  PROC DrawPart102()
    MoveL Offs(pOrigin,206.44,37.94,0.00),v40,z0,tPen\WObj:=wPaper;
    MoveL Offs(pOrigin,207.07,38.36,0.00),v40,z0,tPen\WObj:=wPaper;
    MoveL Offs(pOrigin,206.44,37.94,0.00),v40,fine,tPen\WObj:=wPaper;
    MoveL Offs(pOrigin,206.44,37.94,6.00),v60,z5,tPen\WObj:=wPaper;
    MoveL Offs(pOrigin,207.71,38.79,6.00),vTravel,z5,tPen\WObj:=wPaper;
    MoveL Offs(pOrigin,207.71,38.79,0.00),v60,z0,tPen\WObj:=wPaper;
    MoveL Offs(pOrigin,208.14,39.21,0.00),v40,z0,tPen\WObj:=wPaper;
    MoveL Offs(pOrigin,207.71,38.79,0.00),v40,z0,tPen\WObj:=wPaper;
    MoveL Offs(pOrigin,208.35,39.42,0.00),v40,z0,tPen\WObj:=wPaper;
    MoveL Offs(pOrigin,209.20,40.06,0.00),v40,z0,tPen\WObj:=wPaper;
    MoveL Offs(pOrigin,208.35,39.42,0.00),v40,fine,tPen\WObj:=wPaper;
    MoveL Offs(pOrigin,208.35,39.42,6.00),v60,z5,tPen\WObj:=wPaper;
    MoveL Offs(pOrigin,207.50,40.28,6.00),vTravel,z5,tPen\WObj:=wPaper;
    MoveL Offs(pOrigin,207.50,40.28,0.00),v60,z0,tPen\WObj:=wPaper;
    MoveL Offs(pOrigin,208.14,40.91,0.00),v40,z0,tPen\WObj:=wPaper;
    MoveL Offs(pOrigin,207.50,40.28,0.00),v40,fine,tPen\WObj:=wPaper;
    MoveL Offs(pOrigin,207.50,40.28,6.00),v60,z5,tPen\WObj:=wPaper;
    MoveL Offs(pOrigin,209.41,40.28,6.00),vTravel,z5,tPen\WObj:=wPaper;
    MoveL Offs(pOrigin,209.41,40.28,0.00),v60,z0,tPen\WObj:=wPaper;
    MoveL Offs(pOrigin,209.62,40.70,0.00),v40,z0,tPen\WObj:=wPaper;
    MoveL Offs(pOrigin,209.41,40.28,0.00),v40,fine,tPen\WObj:=wPaper;
    MoveL Offs(pOrigin,209.41,40.28,6.00),v60,z5,tPen\WObj:=wPaper;
    MoveL Offs(pOrigin,209.20,20.51,6.00),vTravel,z5,tPen\WObj:=wPaper;
    MoveL Offs(pOrigin,209.20,20.51,0.00),v60,z0,tPen\WObj:=wPaper;
    MoveL Offs(pOrigin,208.21,19.24,0.00),v40,z0,tPen\WObj:=wPaper;
    MoveL Offs(pOrigin,207.71,17.54,0.00),v40,z0,tPen\WObj:=wPaper;
    MoveL Offs(pOrigin,207.71,16.48,0.00),v40,z0,tPen\WObj:=wPaper;
    MoveL Offs(pOrigin,208.35,14.77,0.00),v40,fine,tPen\WObj:=wPaper;
    MoveL Offs(pOrigin,208.35,14.77,6.00),v60,z5,tPen\WObj:=wPaper;
    MoveL Offs(pOrigin,206.65,19.45,6.00),vTravel,z5,tPen\WObj:=wPaper;
    MoveL Offs(pOrigin,206.65,19.45,0.00),v60,z0,tPen\WObj:=wPaper;
    MoveL Offs(pOrigin,206.86,19.88,0.00),v40,z0,tPen\WObj:=wPaper;
    MoveL Offs(pOrigin,206.65,19.45,0.00),v40,fine,tPen\WObj:=wPaper;
    MoveL Offs(pOrigin,206.65,19.45,6.00),v60,z5,tPen\WObj:=wPaper;
    MoveL Offs(pOrigin,200.49,21.79,6.00),vTravel,z5,tPen\WObj:=wPaper;
    MoveL Offs(pOrigin,200.49,21.79,0.00),v60,z0,tPen\WObj:=wPaper;
    MoveL Offs(pOrigin,206.65,21.36,0.00),v40,z0,tPen\WObj:=wPaper;
    MoveL Offs(pOrigin,207.29,21.08,0.00),v40,z0,tPen\WObj:=wPaper;
    MoveL Offs(pOrigin,206.23,17.96,0.00),v40,z0,tPen\WObj:=wPaper;
    MoveL Offs(pOrigin,206.37,14.85,0.00),v40,z0,tPen\WObj:=wPaper;
    MoveL Offs(pOrigin,205.38,14.85,0.00),v40,z0,tPen\WObj:=wPaper;
    MoveL Offs(pOrigin,204.74,15.41,0.00),v40,z0,tPen\WObj:=wPaper;
    MoveL Offs(pOrigin,196.66,16.48,0.00),v40,z0,tPen\WObj:=wPaper;
    MoveL Offs(pOrigin,195.18,16.40,0.00),v40,z0,tPen\WObj:=wPaper;
    MoveL Offs(pOrigin,194.75,17.33,0.00),v40,z0,tPen\WObj:=wPaper;
    MoveL Offs(pOrigin,194.75,19.45,0.00),v40,z0,tPen\WObj:=wPaper;
    MoveL Offs(pOrigin,195.39,20.87,0.00),v40,z0,tPen\WObj:=wPaper;
    MoveL Offs(pOrigin,196.45,21.15,0.00),v40,z0,tPen\WObj:=wPaper;
    MoveL Offs(pOrigin,196.45,21.15,0.00),v40,z0,tPen\WObj:=wPaper;
    MoveL Offs(pOrigin,196.88,21.58,0.00),v40,z0,tPen\WObj:=wPaper;
    MoveL Offs(pOrigin,197.51,21.58,0.00),v40,z0,tPen\WObj:=wPaper;
    MoveL Offs(pOrigin,197.51,21.58,0.00),v40,z0,tPen\WObj:=wPaper;
    MoveL Offs(pOrigin,198.15,21.15,0.00),v40,z0,tPen\WObj:=wPaper;
    MoveL Offs(pOrigin,200.27,21.15,0.00),v40,z0,tPen\WObj:=wPaper;
    MoveL Offs(pOrigin,200.49,21.79,0.00),v40,z0,tPen\WObj:=wPaper;
    MoveL Offs(pOrigin,200.49,21.79,0.00),v40,z0,tPen\WObj:=wPaper;
    MoveL Offs(pOrigin,197.94,22.00,0.00),v40,z0,tPen\WObj:=wPaper;
    MoveL Offs(pOrigin,197.51,21.58,0.00),v40,z0,tPen\WObj:=wPaper;
    MoveL Offs(pOrigin,196.45,21.15,0.00),v40,z0,tPen\WObj:=wPaper;
    MoveL Offs(pOrigin,195.81,18.60,0.00),v40,z0,tPen\WObj:=wPaper;
    MoveL Offs(pOrigin,196.24,16.48,0.00),v40,fine,tPen\WObj:=wPaper;
    MoveL Offs(pOrigin,196.24,16.48,6.00),v60,z5,tPen\WObj:=wPaper;
    MoveL Offs(pOrigin,157.99,23.27,6.00),vTravel,z5,tPen\WObj:=wPaper;
    MoveL Offs(pOrigin,157.99,23.27,0.00),v60,z0,tPen\WObj:=wPaper;
    MoveL Offs(pOrigin,156.93,23.27,0.00),v40,z0,tPen\WObj:=wPaper;
    MoveL Offs(pOrigin,156.29,23.91,0.00),v40,fine,tPen\WObj:=wPaper;
    MoveL Offs(pOrigin,156.29,23.91,6.00),v60,z5,tPen\WObj:=wPaper;
    MoveL Offs(pOrigin,213.88,70.03,6.00),vTravel,z5,tPen\WObj:=wPaper;
    MoveL Offs(pOrigin,213.88,70.03,0.00),v60,z0,tPen\WObj:=wPaper;
    MoveL Offs(pOrigin,213.66,70.45,0.00),v40,z0,tPen\WObj:=wPaper;
    MoveL Offs(pOrigin,213.88,70.03,0.00),v40,fine,tPen\WObj:=wPaper;
    MoveL Offs(pOrigin,213.88,70.03,6.00),v60,z5,tPen\WObj:=wPaper;
    MoveL Offs(pOrigin,214.94,71.09,6.00),vTravel,z5,tPen\WObj:=wPaper;
    MoveL Offs(pOrigin,214.94,71.09,0.00),v60,z0,tPen\WObj:=wPaper;
    MoveL Offs(pOrigin,214.73,71.51,0.00),v40,z0,tPen\WObj:=wPaper;
    MoveL Offs(pOrigin,214.94,71.09,0.00),v40,fine,tPen\WObj:=wPaper;
    MoveL Offs(pOrigin,214.94,71.09,6.00),v60,z5,tPen\WObj:=wPaper;
    MoveL Offs(pOrigin,214.09,72.57,6.00),vTravel,z5,tPen\WObj:=wPaper;
    MoveL Offs(pOrigin,214.09,72.57,0.00),v60,z0,tPen\WObj:=wPaper;
    MoveL Offs(pOrigin,215.01,71.30,0.00),v40,z0,tPen\WObj:=wPaper;
    MoveL Offs(pOrigin,215.86,68.61,0.00),v40,z0,tPen\WObj:=wPaper;
    MoveL Offs(pOrigin,216.21,68.54,0.00),v40,fine,tPen\WObj:=wPaper;
    MoveL Offs(pOrigin,216.21,68.54,6.00),v60,z5,tPen\WObj:=wPaper;
    MoveL Offs(pOrigin,213.24,73.00,6.00),vTravel,z5,tPen\WObj:=wPaper;
    MoveL Offs(pOrigin,213.24,73.00,0.00),v60,z0,tPen\WObj:=wPaper;
    MoveL Offs(pOrigin,213.52,72.86,0.00),v40,z0,tPen\WObj:=wPaper;
    MoveL Offs(pOrigin,210.90,74.35,0.00),v40,z0,tPen\WObj:=wPaper;
    MoveL Offs(pOrigin,206.86,75.55,0.00),v40,z0,tPen\WObj:=wPaper;
    MoveL Offs(pOrigin,204.10,75.97,0.00),v40,z0,tPen\WObj:=wPaper;
    MoveL Offs(pOrigin,194.96,76.47,0.00),v40,z0,tPen\WObj:=wPaper;
    MoveL Offs(pOrigin,190.50,80.22,0.00),v40,z0,tPen\WObj:=wPaper;
    MoveL Offs(pOrigin,189.86,81.93,0.00),v40,z0,tPen\WObj:=wPaper;
    MoveL Offs(pOrigin,187.74,84.05,0.00),v40,z0,tPen\WObj:=wPaper;
    MoveL Offs(pOrigin,178.03,92.34,0.00),v40,z0,tPen\WObj:=wPaper;
    MoveL Offs(pOrigin,182.14,100.20,0.00),v40,z0,tPen\WObj:=wPaper;
    MoveL Offs(pOrigin,187.74,108.06,0.00),v40,z0,tPen\WObj:=wPaper;
    MoveL Offs(pOrigin,193.26,113.80,0.00),v40,z0,tPen\WObj:=wPaper;
    MoveL Offs(pOrigin,196.24,116.35,0.00),v40,z0,tPen\WObj:=wPaper;
    MoveL Offs(pOrigin,199.64,118.69,0.00),v40,fine,tPen\WObj:=wPaper;
    MoveL Offs(pOrigin,199.64,118.69,6.00),v60,z5,tPen\WObj:=wPaper;
    MoveL Offs(pOrigin,208.14,120.60,6.00),vTravel,z5,tPen\WObj:=wPaper;
    MoveL Offs(pOrigin,208.14,120.60,0.00),v60,z0,tPen\WObj:=wPaper;
    MoveL Offs(pOrigin,207.93,119.32,0.00),v40,z0,tPen\WObj:=wPaper;
    MoveL Offs(pOrigin,209.41,107.64,0.00),v40,z0,tPen\WObj:=wPaper;
    MoveL Offs(pOrigin,210.90,91.06,0.00),v40,fine,tPen\WObj:=wPaper;
    MoveL Offs(pOrigin,210.90,91.06,6.00),v60,z5,tPen\WObj:=wPaper;
    MoveL Offs(pOrigin,195.18,177.34,6.00),vTravel,z5,tPen\WObj:=wPaper;
    MoveL Offs(pOrigin,195.18,177.34,0.00),v60,z0,tPen\WObj:=wPaper;
    MoveL Offs(pOrigin,195.60,177.55,0.00),v40,z0,tPen\WObj:=wPaper;
    MoveL Offs(pOrigin,195.18,177.34,0.00),v40,z0,tPen\WObj:=wPaper;
    MoveL Offs(pOrigin,195.81,177.76,0.00),v40,z0,tPen\WObj:=wPaper;
    MoveL Offs(pOrigin,196.24,177.98,0.00),v40,z0,tPen\WObj:=wPaper;
    MoveL Offs(pOrigin,195.81,177.76,0.00),v40,z0,tPen\WObj:=wPaper;
    MoveL Offs(pOrigin,196.66,178.19,0.00),v40,z0,tPen\WObj:=wPaper;
    MoveL Offs(pOrigin,197.09,178.40,0.00),v40,z0,tPen\WObj:=wPaper;
    MoveL Offs(pOrigin,196.66,178.19,0.00),v40,fine,tPen\WObj:=wPaper;
    MoveL Offs(pOrigin,196.66,178.19,6.00),v60,z5,tPen\WObj:=wPaper;
    MoveL Offs(pOrigin,196.02,179.25,6.00),vTravel,z5,tPen\WObj:=wPaper;
    MoveL Offs(pOrigin,196.02,179.25,0.00),v60,z0,tPen\WObj:=wPaper;
    MoveL Offs(pOrigin,196.45,179.46,0.00),v40,z0,tPen\WObj:=wPaper;
  ENDPROC

  PROC DrawPart103()
    MoveL Offs(pOrigin,196.02,179.25,0.00),v40,z0,tPen\WObj:=wPaper;
    MoveL Offs(pOrigin,195.18,178.82,0.00),v40,z0,tPen\WObj:=wPaper;
    MoveL Offs(pOrigin,195.60,179.04,0.00),v40,z0,tPen\WObj:=wPaper;
    MoveL Offs(pOrigin,195.18,178.82,0.00),v40,fine,tPen\WObj:=wPaper;
    MoveL Offs(pOrigin,195.18,178.82,6.00),v60,z5,tPen\WObj:=wPaper;
    MoveL Offs(pOrigin,194.11,178.19,6.00),vTravel,z5,tPen\WObj:=wPaper;
    MoveL Offs(pOrigin,194.11,178.19,0.00),v60,z0,tPen\WObj:=wPaper;
    MoveL Offs(pOrigin,194.54,178.40,0.00),v40,z0,tPen\WObj:=wPaper;
    MoveL Offs(pOrigin,194.11,178.19,0.00),v40,fine,tPen\WObj:=wPaper;
    MoveL Offs(pOrigin,194.11,178.19,6.00),v60,z5,tPen\WObj:=wPaper;
    MoveL Offs(pOrigin,189.23,181.38,6.00),vTravel,z5,tPen\WObj:=wPaper;
    MoveL Offs(pOrigin,189.23,181.38,0.00),v60,z0,tPen\WObj:=wPaper;
    MoveL Offs(pOrigin,189.86,181.80,0.00),v40,z0,tPen\WObj:=wPaper;
    MoveL Offs(pOrigin,189.86,182.44,0.00),v40,z0,tPen\WObj:=wPaper;
    MoveL Offs(pOrigin,189.86,182.44,0.00),v40,z0,tPen\WObj:=wPaper;
    MoveL Offs(pOrigin,190.07,182.65,0.00),v40,z0,tPen\WObj:=wPaper;
    MoveL Offs(pOrigin,189.86,183.50,0.00),v40,fine,tPen\WObj:=wPaper;
    MoveL Offs(pOrigin,189.86,183.50,6.00),v60,z5,tPen\WObj:=wPaper;
    MoveL Offs(pOrigin,172.86,213.04,6.00),vTravel,z5,tPen\WObj:=wPaper;
    MoveL Offs(pOrigin,172.86,213.04,0.00),v60,z0,tPen\WObj:=wPaper;
    MoveL Offs(pOrigin,172.86,214.31,0.00),v40,z0,tPen\WObj:=wPaper;
    MoveL Offs(pOrigin,173.64,216.86,0.00),v40,z0,tPen\WObj:=wPaper;
    MoveL Offs(pOrigin,175.84,220.69,0.00),v40,z0,tPen\WObj:=wPaper;
    MoveL Offs(pOrigin,178.81,224.09,0.00),v40,z0,tPen\WObj:=wPaper;
    MoveL Offs(pOrigin,182.43,226.64,0.00),v40,z0,tPen\WObj:=wPaper;
    MoveL Offs(pOrigin,182.43,226.64,0.00),v40,z0,tPen\WObj:=wPaper;
    MoveL Offs(pOrigin,183.49,226.64,0.00),v40,z0,tPen\WObj:=wPaper;
    MoveL Offs(pOrigin,183.49,227.27,0.00),v40,z0,tPen\WObj:=wPaper;
    MoveL Offs(pOrigin,183.49,227.27,0.00),v40,z0,tPen\WObj:=wPaper;
    MoveL Offs(pOrigin,184.55,227.42,0.00),v40,z0,tPen\WObj:=wPaper;
    MoveL Offs(pOrigin,189.23,229.47,0.00),v40,z0,tPen\WObj:=wPaper;
    MoveL Offs(pOrigin,194.96,231.31,0.00),v40,z0,tPen\WObj:=wPaper;
    MoveL Offs(pOrigin,200.49,232.59,0.00),v40,z0,tPen\WObj:=wPaper;
    MoveL Offs(pOrigin,202.19,232.66,0.00),v40,z0,tPen\WObj:=wPaper;
    MoveL Offs(pOrigin,202.97,230.04,0.00),v40,z0,tPen\WObj:=wPaper;
    MoveL Offs(pOrigin,204.52,227.91,0.00),v40,z0,tPen\WObj:=wPaper;
    MoveL Offs(pOrigin,206.65,226.85,0.00),v40,z0,tPen\WObj:=wPaper;
    MoveL Offs(pOrigin,208.07,226.85,0.00),v40,z0,tPen\WObj:=wPaper;
    MoveL Offs(pOrigin,209.34,223.66,0.00),v40,z0,tPen\WObj:=wPaper;
    MoveL Offs(pOrigin,211.47,219.84,0.00),v40,z0,tPen\WObj:=wPaper;
    MoveL Offs(pOrigin,215.79,214.74,0.00),v40,z0,tPen\WObj:=wPaper;
    MoveL Offs(pOrigin,216.00,213.89,0.00),v40,z0,tPen\WObj:=wPaper;
    MoveL Offs(pOrigin,207.29,212.61,0.00),v40,z0,tPen\WObj:=wPaper;
    MoveL Offs(pOrigin,201.98,211.20,0.00),v40,z0,tPen\WObj:=wPaper;
    MoveL Offs(pOrigin,197.30,209.28,0.00),v40,z0,tPen\WObj:=wPaper;
    MoveL Offs(pOrigin,181.57,201.28,0.00),v40,z0,tPen\WObj:=wPaper;
    MoveL Offs(pOrigin,174.35,198.30,0.00),v40,z0,tPen\WObj:=wPaper;
    MoveL Offs(pOrigin,172.72,198.02,0.00),v40,z0,tPen\WObj:=wPaper;
    MoveL Offs(pOrigin,170.74,204.32,0.00),v40,z0,tPen\WObj:=wPaper;
    MoveL Offs(pOrigin,169.68,210.49,0.00),v40,z0,tPen\WObj:=wPaper;
    MoveL Offs(pOrigin,169.68,217.50,0.00),v40,z0,tPen\WObj:=wPaper;
    MoveL Offs(pOrigin,170.52,221.54,0.00),v40,z0,tPen\WObj:=wPaper;
    MoveL Offs(pOrigin,172.15,225.57,0.00),v40,z0,tPen\WObj:=wPaper;
    MoveL Offs(pOrigin,173.29,227.27,0.00),v40,z0,tPen\WObj:=wPaper;
    MoveL Offs(pOrigin,175.62,229.61,0.00),v40,z0,tPen\WObj:=wPaper;
    MoveL Offs(pOrigin,179.88,232.02,0.00),v40,z0,tPen\WObj:=wPaper;
    MoveL Offs(pOrigin,183.27,233.30,0.00),v40,z0,tPen\WObj:=wPaper;
    MoveL Offs(pOrigin,183.70,233.86,0.00),v40,z0,tPen\WObj:=wPaper;
    MoveL Offs(pOrigin,183.70,233.86,0.00),v40,z0,tPen\WObj:=wPaper;
    MoveL Offs(pOrigin,186.68,234.50,0.00),v40,fine,tPen\WObj:=wPaper;
    MoveL Offs(pOrigin,186.68,234.50,6.00),v60,z5,tPen\WObj:=wPaper;
    MoveL Offs(pOrigin,183.70,233.86,6.00),vTravel,z5,tPen\WObj:=wPaper;
    MoveL Offs(pOrigin,183.70,233.86,0.00),v60,z0,tPen\WObj:=wPaper;
    MoveL Offs(pOrigin,182.85,234.07,0.00),v40,z0,tPen\WObj:=wPaper;
    MoveL Offs(pOrigin,178.81,232.87,0.00),v40,z0,tPen\WObj:=wPaper;
    MoveL Offs(pOrigin,174.77,230.68,0.00),v40,z0,tPen\WObj:=wPaper;
    MoveL Offs(pOrigin,171.80,227.70,0.00),v40,z0,tPen\WObj:=wPaper;
    MoveL Offs(pOrigin,169.60,223.88,0.00),v40,z0,tPen\WObj:=wPaper;
    MoveL Offs(pOrigin,168.19,217.93,0.00),v40,z0,tPen\WObj:=wPaper;
    MoveL Offs(pOrigin,167.98,212.82,0.00),v40,z0,tPen\WObj:=wPaper;
    MoveL Offs(pOrigin,169.04,205.18,0.00),v40,z0,tPen\WObj:=wPaper;
    MoveL Offs(pOrigin,171.16,197.31,0.00),v40,z0,tPen\WObj:=wPaper;
    MoveL Offs(pOrigin,168.61,196.25,0.00),v40,z0,tPen\WObj:=wPaper;
    MoveL Offs(pOrigin,168.26,196.32,0.00),v40,z0,tPen\WObj:=wPaper;
    MoveL Offs(pOrigin,166.70,202.20,0.00),v40,z0,tPen\WObj:=wPaper;
    MoveL Offs(pOrigin,165.85,209.64,0.00),v40,z0,tPen\WObj:=wPaper;
    MoveL Offs(pOrigin,166.06,216.86,0.00),v40,z0,tPen\WObj:=wPaper;
    MoveL Offs(pOrigin,166.91,221.11,0.00),v40,z0,tPen\WObj:=wPaper;
    MoveL Offs(pOrigin,168.40,224.94,0.00),v40,z0,tPen\WObj:=wPaper;
    MoveL Offs(pOrigin,168.40,225.79,0.00),v40,z0,tPen\WObj:=wPaper;
    MoveL Offs(pOrigin,168.40,225.79,0.00),v40,z0,tPen\WObj:=wPaper;
    MoveL Offs(pOrigin,169.82,227.91,0.00),v40,z0,tPen\WObj:=wPaper;
    MoveL Offs(pOrigin,170.10,229.19,0.00),v40,z0,tPen\WObj:=wPaper;
    MoveL Offs(pOrigin,170.10,229.19,0.00),v40,z0,tPen\WObj:=wPaper;
    MoveL Offs(pOrigin,171.38,230.75,0.00),v40,z0,tPen\WObj:=wPaper;
    MoveL Offs(pOrigin,174.77,232.45,0.00),v40,z0,tPen\WObj:=wPaper;
    MoveL Offs(pOrigin,179.88,234.29,0.00),v40,z0,tPen\WObj:=wPaper;
    MoveL Offs(pOrigin,187.10,236.20,0.00),v40,z0,tPen\WObj:=wPaper;
    MoveL Offs(pOrigin,199.85,238.54,0.00),v40,z0,tPen\WObj:=wPaper;
    MoveL Offs(pOrigin,201.34,238.61,0.00),v40,z0,tPen\WObj:=wPaper;
    MoveL Offs(pOrigin,201.69,238.32,0.00),v40,z0,tPen\WObj:=wPaper;
    MoveL Offs(pOrigin,202.19,235.56,0.00),v40,z0,tPen\WObj:=wPaper;
    MoveL Offs(pOrigin,201.98,233.93,0.00),v40,z0,tPen\WObj:=wPaper;
    MoveL Offs(pOrigin,196.45,232.80,0.00),v40,z0,tPen\WObj:=wPaper;
    MoveL Offs(pOrigin,190.93,231.17,0.00),v40,z0,tPen\WObj:=wPaper;
    MoveL Offs(pOrigin,186.25,229.26,0.00),v40,z0,tPen\WObj:=wPaper;
    MoveL Offs(pOrigin,183.49,227.70,0.00),v40,z0,tPen\WObj:=wPaper;
    MoveL Offs(pOrigin,183.49,227.70,0.00),v40,z0,tPen\WObj:=wPaper;
    MoveL Offs(pOrigin,182.85,227.49,0.00),v40,z0,tPen\WObj:=wPaper;
    MoveL Offs(pOrigin,182.43,226.64,0.00),v40,fine,tPen\WObj:=wPaper;
    MoveL Offs(pOrigin,182.43,226.64,6.00),v60,z5,tPen\WObj:=wPaper;
    MoveL Offs(pOrigin,184.12,228.34,6.00),vTravel,z5,tPen\WObj:=wPaper;
    MoveL Offs(pOrigin,184.12,228.34,0.00),v60,z0,tPen\WObj:=wPaper;
    MoveL Offs(pOrigin,184.55,228.55,0.00),v40,z0,tPen\WObj:=wPaper;
    MoveL Offs(pOrigin,184.12,228.34,0.00),v40,fine,tPen\WObj:=wPaper;
    MoveL Offs(pOrigin,184.12,228.34,6.00),v60,z5,tPen\WObj:=wPaper;
    MoveL Offs(pOrigin,186.89,229.61,6.00),vTravel,z5,tPen\WObj:=wPaper;
    MoveL Offs(pOrigin,186.89,229.61,0.00),v60,z0,tPen\WObj:=wPaper;
    MoveL Offs(pOrigin,187.31,229.82,0.00),v40,z0,tPen\WObj:=wPaper;
    MoveL Offs(pOrigin,186.89,229.61,0.00),v40,fine,tPen\WObj:=wPaper;
    MoveL Offs(pOrigin,186.89,229.61,6.00),v60,z5,tPen\WObj:=wPaper;
    MoveL Offs(pOrigin,177.96,232.59,6.00),vTravel,z5,tPen\WObj:=wPaper;
    MoveL Offs(pOrigin,177.96,232.59,0.00),v60,z0,tPen\WObj:=wPaper;
    MoveL Offs(pOrigin,178.39,232.80,0.00),v40,z0,tPen\WObj:=wPaper;
    MoveL Offs(pOrigin,177.96,232.59,0.00),v40,fine,tPen\WObj:=wPaper;
    MoveL Offs(pOrigin,177.96,232.59,6.00),v60,z5,tPen\WObj:=wPaper;
    MoveL Offs(pOrigin,174.35,230.46,6.00),vTravel,z5,tPen\WObj:=wPaper;
    MoveL Offs(pOrigin,174.35,230.46,0.00),v60,z0,tPen\WObj:=wPaper;
    MoveL Offs(pOrigin,174.77,230.89,0.00),v40,z0,tPen\WObj:=wPaper;
    MoveL Offs(pOrigin,174.35,230.46,0.00),v40,z0,tPen\WObj:=wPaper;
  ENDPROC

  PROC DrawPart104()
    MoveL Offs(pOrigin,173.71,230.04,0.00),v40,z0,tPen\WObj:=wPaper;
    MoveL Offs(pOrigin,174.14,230.25,0.00),v40,z0,tPen\WObj:=wPaper;
    MoveL Offs(pOrigin,173.71,230.04,0.00),v40,fine,tPen\WObj:=wPaper;
    MoveL Offs(pOrigin,173.71,230.04,6.00),v60,z5,tPen\WObj:=wPaper;
    MoveL Offs(pOrigin,175.20,228.98,6.00),vTravel,z5,tPen\WObj:=wPaper;
    MoveL Offs(pOrigin,175.20,228.98,0.00),v60,z0,tPen\WObj:=wPaper;
    MoveL Offs(pOrigin,175.84,229.61,0.00),v40,z0,tPen\WObj:=wPaper;
    MoveL Offs(pOrigin,175.20,228.98,0.00),v40,fine,tPen\WObj:=wPaper;
    MoveL Offs(pOrigin,175.20,228.98,6.00),v60,z5,tPen\WObj:=wPaper;
    MoveL Offs(pOrigin,173.71,227.49,6.00),vTravel,z5,tPen\WObj:=wPaper;
    MoveL Offs(pOrigin,173.71,227.49,0.00),v60,z0,tPen\WObj:=wPaper;
    MoveL Offs(pOrigin,174.56,228.34,0.00),v40,z0,tPen\WObj:=wPaper;
    MoveL Offs(pOrigin,173.71,227.49,0.00),v40,fine,tPen\WObj:=wPaper;
    MoveL Offs(pOrigin,173.71,227.49,6.00),v60,z5,tPen\WObj:=wPaper;
    MoveL Offs(pOrigin,172.01,228.12,6.00),vTravel,z5,tPen\WObj:=wPaper;
    MoveL Offs(pOrigin,172.01,228.12,0.00),v60,z0,tPen\WObj:=wPaper;
    MoveL Offs(pOrigin,172.65,228.76,0.00),v40,z0,tPen\WObj:=wPaper;
    MoveL Offs(pOrigin,172.01,228.12,0.00),v40,fine,tPen\WObj:=wPaper;
    MoveL Offs(pOrigin,172.01,228.12,6.00),v60,z5,tPen\WObj:=wPaper;
    MoveL Offs(pOrigin,170.10,229.19,6.00),vTravel,z5,tPen\WObj:=wPaper;
    MoveL Offs(pOrigin,170.10,229.19,0.00),v60,z0,tPen\WObj:=wPaper;
    MoveL Offs(pOrigin,168.82,228.76,0.00),v40,z0,tPen\WObj:=wPaper;
    MoveL Offs(pOrigin,165.43,224.94,0.00),v40,z0,tPen\WObj:=wPaper;
    MoveL Offs(pOrigin,163.23,220.90,0.00),v40,z0,tPen\WObj:=wPaper;
    MoveL Offs(pOrigin,162.24,217.50,0.00),v40,z0,tPen\WObj:=wPaper;
    MoveL Offs(pOrigin,161.60,213.89,0.00),v40,z0,tPen\WObj:=wPaper;
    MoveL Offs(pOrigin,161.18,208.15,0.00),v40,z0,tPen\WObj:=wPaper;
    MoveL Offs(pOrigin,161.18,194.55,0.00),v40,z0,tPen\WObj:=wPaper;
    MoveL Offs(pOrigin,161.60,194.12,0.00),v40,z0,tPen\WObj:=wPaper;
    MoveL Offs(pOrigin,166.27,195.47,0.00),v40,z0,tPen\WObj:=wPaper;
    MoveL Offs(pOrigin,166.70,196.04,0.00),v40,z0,tPen\WObj:=wPaper;
    MoveL Offs(pOrigin,164.79,204.96,0.00),v40,z0,tPen\WObj:=wPaper;
    MoveL Offs(pOrigin,164.36,209.21,0.00),v40,z0,tPen\WObj:=wPaper;
    MoveL Offs(pOrigin,164.36,214.10,0.00),v40,z0,tPen\WObj:=wPaper;
    MoveL Offs(pOrigin,164.79,217.71,0.00),v40,z0,tPen\WObj:=wPaper;
    MoveL Offs(pOrigin,165.78,221.54,0.00),v40,z0,tPen\WObj:=wPaper;
    MoveL Offs(pOrigin,167.48,225.36,0.00),v40,z0,tPen\WObj:=wPaper;
    MoveL Offs(pOrigin,168.40,225.79,0.00),v40,fine,tPen\WObj:=wPaper;
    MoveL Offs(pOrigin,168.40,225.79,6.00),v60,z5,tPen\WObj:=wPaper;
    MoveL Offs(pOrigin,166.70,226.85,6.00),vTravel,z5,tPen\WObj:=wPaper;
    MoveL Offs(pOrigin,166.70,226.85,0.00),v60,z0,tPen\WObj:=wPaper;
    MoveL Offs(pOrigin,168.82,228.98,0.00),v40,z0,tPen\WObj:=wPaper;
    MoveL Offs(pOrigin,166.70,226.85,0.00),v40,z0,tPen\WObj:=wPaper;
    MoveL Offs(pOrigin,166.06,226.00,0.00),v40,z0,tPen\WObj:=wPaper;
    MoveL Offs(pOrigin,166.49,226.43,0.00),v40,z0,tPen\WObj:=wPaper;
    MoveL Offs(pOrigin,166.06,226.00,0.00),v40,fine,tPen\WObj:=wPaper;
    MoveL Offs(pOrigin,166.06,226.00,6.00),v60,z5,tPen\WObj:=wPaper;
    MoveL Offs(pOrigin,164.36,226.43,6.00),vTravel,z5,tPen\WObj:=wPaper;
    MoveL Offs(pOrigin,164.36,226.43,0.00),v60,z0,tPen\WObj:=wPaper;
    MoveL Offs(pOrigin,165.21,227.49,0.00),v40,z0,tPen\WObj:=wPaper;
    MoveL Offs(pOrigin,164.36,226.43,0.00),v40,fine,tPen\WObj:=wPaper;
    MoveL Offs(pOrigin,164.36,226.43,6.00),v60,z5,tPen\WObj:=wPaper;
    MoveL Offs(pOrigin,165.00,224.51,6.00),vTravel,z5,tPen\WObj:=wPaper;
    MoveL Offs(pOrigin,165.00,224.51,0.00),v60,z0,tPen\WObj:=wPaper;
    MoveL Offs(pOrigin,165.21,224.94,0.00),v40,z0,tPen\WObj:=wPaper;
    MoveL Offs(pOrigin,165.00,224.51,0.00),v40,fine,tPen\WObj:=wPaper;
    MoveL Offs(pOrigin,165.00,224.51,6.00),v60,z5,tPen\WObj:=wPaper;
    MoveL Offs(pOrigin,164.15,223.02,6.00),vTravel,z5,tPen\WObj:=wPaper;
    MoveL Offs(pOrigin,164.15,223.02,0.00),v60,z0,tPen\WObj:=wPaper;
    MoveL Offs(pOrigin,164.36,223.45,0.00),v40,z0,tPen\WObj:=wPaper;
    MoveL Offs(pOrigin,164.15,223.02,0.00),v40,fine,tPen\WObj:=wPaper;
    MoveL Offs(pOrigin,164.15,223.02,6.00),v60,z5,tPen\WObj:=wPaper;
    MoveL Offs(pOrigin,163.09,224.51,6.00),vTravel,z5,tPen\WObj:=wPaper;
    MoveL Offs(pOrigin,163.09,224.51,0.00),v60,z0,tPen\WObj:=wPaper;
    MoveL Offs(pOrigin,163.30,224.94,0.00),v40,z0,tPen\WObj:=wPaper;
    MoveL Offs(pOrigin,163.09,224.51,0.00),v40,fine,tPen\WObj:=wPaper;
    MoveL Offs(pOrigin,163.09,224.51,6.00),v60,z5,tPen\WObj:=wPaper;
    MoveL Offs(pOrigin,162.24,222.81,6.00),vTravel,z5,tPen\WObj:=wPaper;
    MoveL Offs(pOrigin,162.24,222.81,0.00),v60,z0,tPen\WObj:=wPaper;
    MoveL Offs(pOrigin,162.45,223.24,0.00),v40,z0,tPen\WObj:=wPaper;
    MoveL Offs(pOrigin,162.24,222.81,0.00),v40,fine,tPen\WObj:=wPaper;
    MoveL Offs(pOrigin,162.24,222.81,6.00),v60,z5,tPen\WObj:=wPaper;
    MoveL Offs(pOrigin,166.70,223.45,6.00),vTravel,z5,tPen\WObj:=wPaper;
    MoveL Offs(pOrigin,166.70,223.45,0.00),v60,z0,tPen\WObj:=wPaper;
    MoveL Offs(pOrigin,166.91,223.88,0.00),v40,z0,tPen\WObj:=wPaper;
    MoveL Offs(pOrigin,166.70,223.45,0.00),v40,fine,tPen\WObj:=wPaper;
    MoveL Offs(pOrigin,166.70,223.45,6.00),v60,z5,tPen\WObj:=wPaper;
    MoveL Offs(pOrigin,171.80,224.51,6.00),vTravel,z5,tPen\WObj:=wPaper;
    MoveL Offs(pOrigin,171.80,224.51,0.00),v60,z0,tPen\WObj:=wPaper;
    MoveL Offs(pOrigin,172.01,224.94,0.00),v40,z0,tPen\WObj:=wPaper;
    MoveL Offs(pOrigin,171.80,224.51,0.00),v40,fine,tPen\WObj:=wPaper;
    MoveL Offs(pOrigin,171.80,224.51,6.00),v60,z5,tPen\WObj:=wPaper;
    MoveL Offs(pOrigin,166.49,228.98,6.00),vTravel,z5,tPen\WObj:=wPaper;
    MoveL Offs(pOrigin,166.49,228.98,0.00),v60,z0,tPen\WObj:=wPaper;
    MoveL Offs(pOrigin,166.91,229.40,0.00),v40,z0,tPen\WObj:=wPaper;
    MoveL Offs(pOrigin,166.49,228.98,0.00),v40,fine,tPen\WObj:=wPaper;
    MoveL Offs(pOrigin,166.49,228.98,6.00),v60,z5,tPen\WObj:=wPaper;
    MoveL Offs(pOrigin,169.04,231.10,6.00),vTravel,z5,tPen\WObj:=wPaper;
    MoveL Offs(pOrigin,169.04,231.10,0.00),v60,z0,tPen\WObj:=wPaper;
    MoveL Offs(pOrigin,169.68,231.52,0.00),v40,z0,tPen\WObj:=wPaper;
    MoveL Offs(pOrigin,169.04,231.10,0.00),v40,fine,tPen\WObj:=wPaper;
    MoveL Offs(pOrigin,169.04,231.10,6.00),v60,z5,tPen\WObj:=wPaper;
    MoveL Offs(pOrigin,170.74,232.16,6.00),vTravel,z5,tPen\WObj:=wPaper;
    MoveL Offs(pOrigin,170.74,232.16,0.00),v60,z0,tPen\WObj:=wPaper;
    MoveL Offs(pOrigin,171.16,232.38,0.00),v40,z0,tPen\WObj:=wPaper;
    MoveL Offs(pOrigin,170.74,232.16,0.00),v40,z0,tPen\WObj:=wPaper;
    MoveL Offs(pOrigin,171.59,232.59,0.00),v40,z0,tPen\WObj:=wPaper;
    MoveL Offs(pOrigin,172.23,233.01,0.00),v40,z0,tPen\WObj:=wPaper;
    MoveL Offs(pOrigin,171.59,232.59,0.00),v40,fine,tPen\WObj:=wPaper;
    MoveL Offs(pOrigin,171.59,232.59,6.00),v60,z5,tPen\WObj:=wPaper;
    MoveL Offs(pOrigin,173.71,233.65,6.00),vTravel,z5,tPen\WObj:=wPaper;
    MoveL Offs(pOrigin,173.71,233.65,0.00),v60,z0,tPen\WObj:=wPaper;
    MoveL Offs(pOrigin,174.14,233.86,0.00),v40,z0,tPen\WObj:=wPaper;
    MoveL Offs(pOrigin,173.71,233.65,0.00),v40,fine,tPen\WObj:=wPaper;
    MoveL Offs(pOrigin,173.71,233.65,6.00),v60,z5,tPen\WObj:=wPaper;
    MoveL Offs(pOrigin,230.88,186.69,6.00),vTravel,z5,tPen\WObj:=wPaper;
    MoveL Offs(pOrigin,230.88,186.69,0.00),v60,z0,tPen\WObj:=wPaper;
    MoveL Offs(pOrigin,231.30,187.11,0.00),v40,z0,tPen\WObj:=wPaper;
    MoveL Offs(pOrigin,230.88,186.69,0.00),v40,fine,tPen\WObj:=wPaper;
    MoveL Offs(pOrigin,230.88,186.69,6.00),v60,z5,tPen\WObj:=wPaper;
    MoveL Offs(pOrigin,407.25,41.34,6.00),vTravel,z5,tPen\WObj:=wPaper;
    MoveL Offs(pOrigin,407.25,41.34,0.00),v60,z0,tPen\WObj:=wPaper;
    MoveL Offs(pOrigin,407.46,41.76,0.00),v40,z0,tPen\WObj:=wPaper;
    MoveL Offs(pOrigin,407.25,41.34,0.00),v40,fine,tPen\WObj:=wPaper;
    MoveL Offs(pOrigin,407.25,41.34,6.00),v60,z5,tPen\WObj:=wPaper;
    MoveL Offs(pOrigin,409.59,40.70,6.00),vTravel,z5,tPen\WObj:=wPaper;
    MoveL Offs(pOrigin,409.59,40.70,0.00),v60,z0,tPen\WObj:=wPaper;
    MoveL Offs(pOrigin,410.44,41.55,0.00),v40,z0,tPen\WObj:=wPaper;
    MoveL Offs(pOrigin,409.59,40.70,0.00),v40,fine,tPen\WObj:=wPaper;
    MoveL Offs(pOrigin,409.59,40.70,6.00),v60,z5,tPen\WObj:=wPaper;
  ENDPROC

  PROC DrawPart105()
    MoveL Offs(pOrigin,410.86,41.76,6.00),vTravel,z5,tPen\WObj:=wPaper;
    MoveL Offs(pOrigin,410.86,41.76,0.00),v60,z0,tPen\WObj:=wPaper;
    MoveL Offs(pOrigin,411.71,42.61,0.00),v40,z0,tPen\WObj:=wPaper;
    MoveL Offs(pOrigin,410.86,41.76,0.00),v40,fine,tPen\WObj:=wPaper;
    MoveL Offs(pOrigin,410.86,41.76,6.00),v60,z5,tPen\WObj:=wPaper;
  ENDPROC

ENDMODULE
